// TIA Portal V21 export
ORGANIZATION_BLOCK "Main"   // OB1, LAD, ProgramCycle
TITLE = "Main Program Sweep (Cycle)"
{ S7_Optimized_Access := 'TRUE' }
// stored: SetENOAutomatically false
   VAR_INPUT
      Initial_Call : Bool;   // Initial call of this OB
      Remanence : Bool;   // =True, if remanent data are available
   END_VAR
   VAR_TEMP   // added for the SCL form of the ladder/FBD networks
      _w1 : Bool;
   END_VAR
BEGIN

REGION Network 1: "Sec_Pulse"
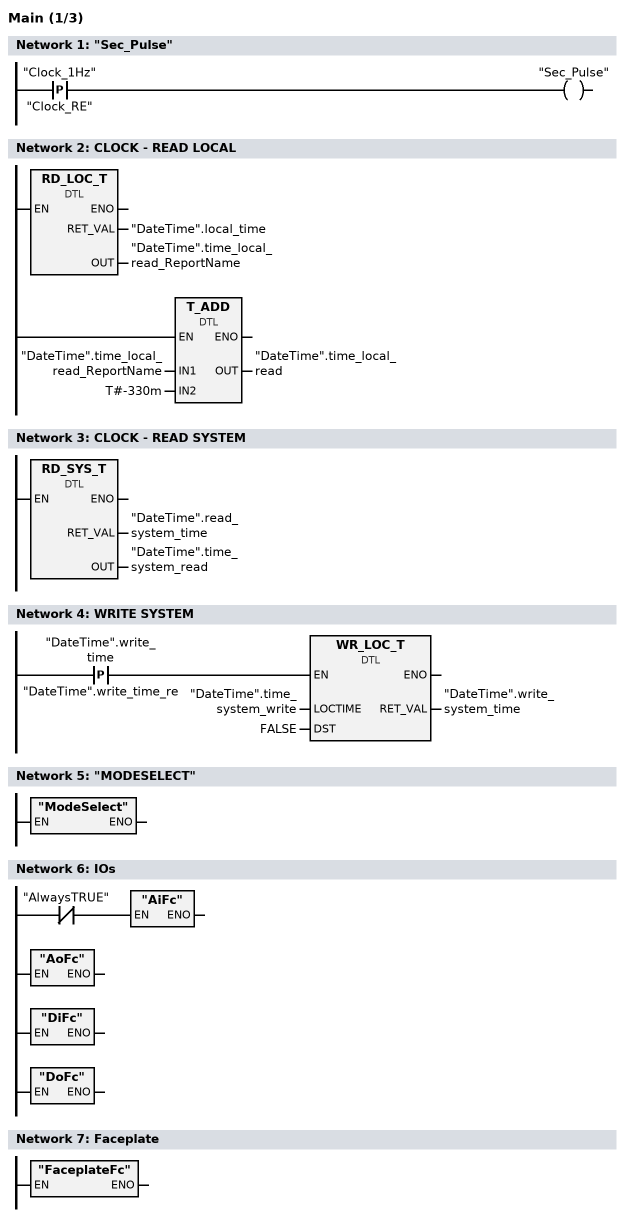
   RUNG wire#powerrail
      P_Contact(operand := "Clock_1Hz", bit := "Clock_RE")
      Coil( "Sec_Pulse" )
   END_RUNG
   // the same network as SCL:
   #_w1 := "Clock_1Hz" AND NOT "Clock_RE";   // rising edge of "Clock_1Hz"
   "Clock_RE" := "Clock_1Hz";
   "Sec_Pulse" := #_w1;
END_REGION

REGION Network 2: CLOCK - READ LOCAL
   RUNG wire#powerrail
      { S7_Templates := "date_type := DTL" } RD_LOC_T(RET_VAL => "DateTime".local_time, OUT => "DateTime".time_local_read_ReportName)
   END_RUNG
   RUNG wire#powerrail
      { S7_Templates := "[date_type := DTL, time_type := Time]" } T_ADD(IN1 := "DateTime".time_local_read_ReportName, IN2 := T#-330m, OUT => "DateTime".time_local_read)
   END_RUNG
   // the same network as SCL:
   "DateTime".local_time := RD_LOC_T(OUT => "DateTime".time_local_read_ReportName);
   T_ADD(IN1 := "DateTime".time_local_read_ReportName, IN2 := T#-330m, OUT => "DateTime".time_local_read);
END_REGION

REGION Network 3: CLOCK - READ SYSTEM
   RUNG wire#powerrail
      { S7_Templates := "date_type := DTL" } RD_SYS_T(RET_VAL => "DateTime".read_system_time, OUT => "DateTime".time_system_read)
   END_RUNG
   // the same network as SCL:
   "DateTime".read_system_time := RD_SYS_T(OUT => "DateTime".time_system_read);
END_REGION

REGION Network 4: WRITE SYSTEM
   RUNG wire#powerrail
      P_Contact(operand := "DateTime".write_time, bit := "DateTime".write_time_re)
      { S7_Templates := "loctime_type := DTL" } WR_LOC_T(LOCTIME := "DateTime".time_system_write, DST := FALSE, Ret_Val => "DateTime".write_system_time)
   END_RUNG
   // the same network as SCL:
   #_w1 := "DateTime".write_time AND NOT "DateTime".write_time_re;   // rising edge of "DateTime".write_time
   "DateTime".write_time_re := "DateTime".write_time;
   IF #_w1 THEN
       "DateTime".write_system_time := WR_LOC_T(LOCTIME := "DateTime".time_system_write, DST := FALSE);
   END_IF;
END_REGION

REGION Network 5: "MODESELECT"
   RUNG wire#powerrail
      "ModeSelect"()
   END_RUNG
   // the same network as SCL:
   "ModeSelect"();
END_REGION

REGION Network 6: IOs
   RUNG wire#powerrail
      I_Contact( "AlwaysTRUE" )
      "AiFc"()
   END_RUNG
   RUNG wire#powerrail
      "AoFc"()
   END_RUNG
   RUNG wire#powerrail
      "DiFc"()
   END_RUNG
   RUNG wire#powerrail
      "DoFc"()
   END_RUNG
   // the same network as SCL:
   IF NOT "AlwaysTRUE" THEN "AiFc"(); END_IF;
   "AoFc"();
   "DiFc"();
   "DoFc"();
END_REGION

REGION Network 7: Faceplate
   RUNG wire#powerrail
      "FaceplateFc"()
   END_RUNG
   // the same network as SCL:
   "FaceplateFc"();
END_REGION

REGION Network 8: ValvesOutputFc
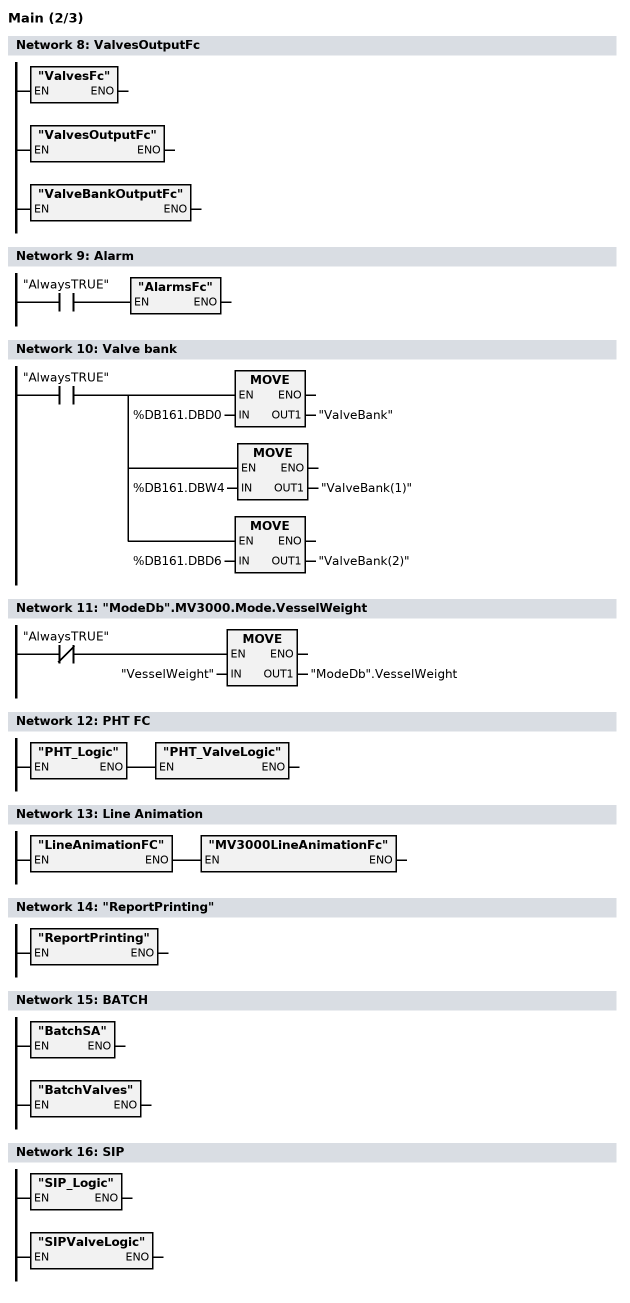
   RUNG wire#powerrail
      "ValvesFc"()
   END_RUNG
   RUNG wire#powerrail
      "ValvesOutputFc"()
   END_RUNG
   RUNG wire#powerrail
      "ValveBankOutputFc"()
   END_RUNG
   // the same network as SCL:
   "ValvesFc"();
   "ValvesOutputFc"();
   "ValveBankOutputFc"();
END_REGION

REGION Network 9: Alarm
   RUNG wire#powerrail
      Contact( "AlwaysTRUE" )
      "AlarmsFc"()
   END_RUNG
   // the same network as SCL:
   IF "AlwaysTRUE" THEN "AlarmsFc"(); END_IF;
END_REGION

REGION Network 10: Valve bank
   RUNG wire#powerrail
      Contact( "AlwaysTRUE" )
      wire#w1
      Move(in := %DB161.DBD0, out1 => "ValveBank")
   END_RUNG
   RUNG wire#w1
      Move(in := %DB161.DBW4, out1 => "ValveBank(1)")
   END_RUNG
   RUNG wire#w1
      Move(in := %DB161.DBD6, out1 => "ValveBank(2)")
   END_RUNG
   // the same network as SCL:
   IF "AlwaysTRUE" THEN
       "ValveBank" := %DB161.DBD0;
       "ValveBank(1)" := %DB161.DBW4;
       "ValveBank(2)" := %DB161.DBD6;
   END_IF;
END_REGION

REGION Network 11: "ModeDb".MV3000.Mode.VesselWeight
   RUNG wire#powerrail
      I_Contact( "AlwaysTRUE" )
      Move(in := "VesselWeight", out1 => "ModeDb".VesselWeight)
   END_RUNG
   // the same network as SCL:
   IF NOT "AlwaysTRUE" THEN "ModeDb".VesselWeight := "VesselWeight"; END_IF;
END_REGION

REGION Network 12: PHT FC
   RUNG wire#powerrail
      "PHT_Logic"()
      "PHT_ValveLogic"()
   END_RUNG
   // the same network as SCL:
   "PHT_Logic"(ENO => #_w1);
   IF #_w1 THEN "PHT_ValveLogic"(); END_IF;
END_REGION

REGION Network 13: Line Animation
   RUNG wire#powerrail
      "LineAnimationFC"()
      "MV3000LineAnimationFc"()
   END_RUNG
   // the same network as SCL:
   "LineAnimationFC"(ENO => #_w1);
   IF #_w1 THEN "MV3000LineAnimationFc"(); END_IF;
END_REGION

REGION Network 14: "ReportPrinting"
   RUNG wire#powerrail
      "ReportPrinting"()
   END_RUNG
   // the same network as SCL:
   "ReportPrinting"();
END_REGION

REGION Network 15: BATCH
   RUNG wire#powerrail
      "BatchSA"()
   END_RUNG
   RUNG wire#powerrail
      "BatchValves"()
   END_RUNG
   // the same network as SCL:
   "BatchSA"();
   "BatchValves"();
END_REGION

REGION Network 16: SIP
   RUNG wire#powerrail
      "SIP_Logic"()
   END_RUNG
   RUNG wire#powerrail
      "SIPValveLogic"()
   END_RUNG
   // the same network as SCL:
   "SIP_Logic"();
   "SIPValveLogic"();
END_REGION

REGION Network 17: CIP
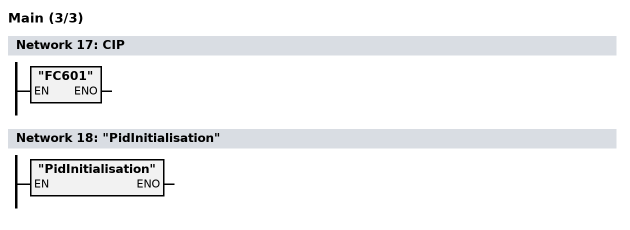
   RUNG wire#powerrail
      "FC601"()
   END_RUNG
   // the same network as SCL:
   "FC601"();
END_REGION

REGION Network 18: "PidInitialisation"
   RUNG wire#powerrail
      "PidInitialisation"()
   END_RUNG
   // the same network as SCL:
   "PidInitialisation"();
END_REGION
END_ORGANIZATION_BLOCK
